// TwinCAT 3 PLC project BohrMachine
// ProgramVersion: 3.1.4023.0
// libraries:
//   Tc2_MC2, * (Beckhoff Automation GmbH)
//   Tc2_Standard, * (Beckhoff Automation GmbH)
//   Tc2_System, * (Beckhoff Automation GmbH)
//   Tc2_Utilities, * (Beckhoff Automation GmbH)
//   Tc3_EventLogger, * (Beckhoff Automation GmbH)
//   Tc3_Module, * (Beckhoff Automation GmbH)
//   VisuSymbols,3.5.10.0,System
// project tree:
//   DUTs/ E_BOHRER_STATES.TcDUT
//   / GlobalTextList.TcGTLO, PlcTask.TcTTO, VisualizationManager.TcVMO (not stored)
//   GVLs/ GVL_Config.TcGVL, GVL_Control.TcGVL
//   POUs/ AxesManager.TcPOU, Bohrkopf.TcPOU, Bohrmaschine.TcPOU, F_Log.TcPOU, I_MachineLogger.TcIO, MachineLogger.TcPOU, MAIN.TcPOU
//   VISUs/ UI.TcVIS
// real-time tasks:
//   TASK PlcTask: cycle T#10ms, priority 20, ADS port 350
//   TASK PlcTask1: cycle T#10ms, priority 21, ADS port 351
//   TASK PlcTask2: cycle T#10ms, priority 22, ADS port 352
//   TASK PlcTask3: cycle T#10ms, priority 23, ADS port 353
//   TASK ControllerTask: cycle T#10ms, priority 1, ADS port 354
//   TASK PlcTask4: cycle T#10ms, priority 24, ADS port 355
//   TASK PlcTask5: cycle T#10ms, priority 25, ADS port 356
// motion (NC):
//   TASK NC-Task 1 SAF: cycle T#2ms, priority 4, ADS port 501
//   TASK NC-Task 1 SVB: cycle T#10ms, priority 8, ADS port 511
//   AXIS xAchse (id 1) // Links-Rechts-Bewegung des Bohrers
//     OtherSettings: AllowMotionCmdToSlave=true
//     encoder EncType=1
//     drive DrvType=5
//       Analog: TorqueSetpointScale=10
//       TimeComp: TaskDelayCycles=1
//     controller CtrType=1
//       CtrPara: PriorControlFactor=1
//         Observer: BandWidth=20
//   AXIS yAchse (id 2) // Hoch-Runter-Bewegung des Bohrers
//     OtherSettings: AllowMotionCmdToSlave=true
//     encoder EncType=1
//     drive DrvType=5
//       Analog: TorqueSetpointScale=10
//       TimeComp: TaskDelayCycles=1
//     controller CtrType=1
//       CtrPara: PriorControlFactor=1
//         Observer: BandWidth=20
//   AXIS zAchse (id 3) // Vor-Zurück-Bewegung des Bohrers
//     OtherSettings: AllowMotionCmdToSlave=true
//     encoder EncType=1
//     drive DrvType=5
//       Analog: TorqueSetpointScale=10
//       TimeComp: TaskDelayCycles=1
//     controller CtrType=1
//       CtrPara: PriorControlFactor=1
//         Observer: BandWidth=20
//   AXIS TransportA (id 4)
//     OtherSettings: AllowMotionCmdToSlave=true
//     encoder EncType=1
//     drive DrvType=5
//       Analog: TorqueSetpointScale=10
//       TimeComp: TaskDelayCycles=1
//     controller CtrType=1
//       CtrPara: PriorControlFactor=1
//         Observer: BandWidth=20
//   AXIS TransportB (id 5)
//     OtherSettings: AllowMotionCmdToSlave=true
//     encoder EncType=1
//     drive DrvType=5
//       Analog: TorqueSetpointScale=10
//       TimeComp: TaskDelayCycles=1
//     controller CtrType=1
//       CtrPara: PriorControlFactor=1
//         Observer: BandWidth=20
// variable links:
//   BohrMachine/BohrMachine Instance <-> Controller/Controller_Obj1 (ModuleController)
//     PlcTask Outputs/MAIN.bohrmaschine.eZustand <-> Bohrmaschine/State
//     PlcTask Outputs/MAIN.bohrmaschine.objID <-> InputIPointers/oidBohrmaschine
//   SuperBohrmachine/SuperBohrmachine Instance <-> NC-Task 1 SAF/Axes/xAchse
//     PlcTask Inputs/MAIN.fbSuperBohrmachine.fbAxesManager.xAchse.NcToPlc <-> Outputs/ToPlc
//     PlcTask Outputs/MAIN.fbSuperBohrmachine.fbAxesManager.xAchse.PlcToNc <-> Inputs/FromPlc
//   SuperBohrmachine/SuperBohrmachine Instance <-> NC-Task 1 SAF/Axes/yAchse
//     PlcTask Inputs/MAIN.fbSuperBohrmachine.fbBohrkopf.axisRef.NcToPlc <-> Outputs/ToPlc
//     PlcTask Outputs/MAIN.fbSuperBohrmachine.fbBohrkopf.axisRef.PlcToNc <-> Inputs/FromPlc
//   SuperBohrmachine/SuperBohrmachine Instance <-> NC-Task 1 SAF/Axes/zAchse
//     PlcTask Inputs/MAIN.fbSuperBohrmachine.fbAxesManager.zAchse.NcToPlc <-> Outputs/ToPlc
//     PlcTask Outputs/MAIN.fbSuperBohrmachine.fbAxesManager.zAchse.PlcToNc <-> Inputs/FromPlc
//   TransportA/TransportA Instance <-> NC-Task 1 SAF/Axes/TransportA
//     PlcTask Inputs/MAIN.fbTransport.axisTransportA.NcToPlc <-> Outputs/ToPlc
//     PlcTask Outputs/MAIN.fbTransport.axisTransportA.PlcToNc <-> Inputs/FromPlc
//   TransportA/TransportA Instance <-> TransportB/TransportB Instance
//     PlcTask Outputs/MAIN.fbTransport.rActVelocity <-> PlcTask Inputs/MAIN.fbTransportSlave.rMasterVelocity
//   TransportA/TransportA Instance <-> Controller/Controller_Obj1 (ModuleController)
//     PlcTask Outputs/MAIN.fbTransport.eZustand <-> TransportA/State
//     PlcTask Outputs/MAIN.fbTransport.objID <-> InputIPointers/oidTransportA
//   TransportB/TransportB Instance <-> NC-Task 1 SAF/Axes/TransportB
//     PlcTask Inputs/MAIN.fbTransportSlave.axisTransportB.NcToPlc <-> Outputs/ToPlc
//     PlcTask Outputs/MAIN.fbTransportSlave.axisTransportB.PlcToNc <-> Inputs/FromPlc
//   TransportB/TransportB Instance <-> Controller/Controller_Obj1 (ModuleController)
//     PlcTask Outputs/MAIN.fbTransportSlave.eZustand <-> TransportB/State
//     PlcTask Outputs/MAIN.fbTransportSlave.fbSensor.bWerkStueckLiegtAn <-> TransportB/WerkstueckLiegtAn
//     PlcTask Outputs/MAIN.fbTransportSlave.objID <-> InputIPointers/oidTransportB

CONFIGURATION BohrMachine
    RESOURCE PLC ON TwinCAT3
        TASK PlcTask(INTERVAL := T#10ms, PRIORITY := 20);
        PROGRAM MAIN WITH PlcTask : MAIN;
    END_RESOURCE
END_CONFIGURATION

// ---- DUTs/E_BOHRER_STATES.TcDUT
{attribute 'qualified_only'}
{attribute 'strict'}
TYPE E_BOHRER_STATES :
(
	eBereit := 0,
	eHerunterfahrend,
	eHochfahrend,
	eUnten,
	eOben,
	eFertig
);
END_TYPE

// ---- GVLs/GVL_Config.TcGVL
{attribute 'qualified_only'}
VAR_GLOBAL
	// Konfiguration
//	stConfig: ST_Config := (rLaenge := 400, rBreite := 300, rDicke := 30);
END_VAR

// ---- GVLs/GVL_Control.TcGVL
{attribute 'qualified_only'}
VAR_GLOBAL
	// UI Command
	bRun: BOOL := FALSE;
	// UI Indicator
	bIsRunning: BOOL := FALSE;
	nProgress: USINT := 0;
	
	// bErrors: BOOL := FALSE;
END_VAR

// ---- POUs/I_MachineLogger.TcIO
INTERFACE I_MachineLogger

METHOD LogBohrung : BOOL
VAR_INPUT
	stPunkt: REFERENCE TO ST_2DPoint;
END_VAR
END_METHOD

METHOD LogPunktAngefahren : BOOL
VAR_INPUT
	stPunkt: REFERENCE TO ST_2DPoint;
END_VAR
END_METHOD

METHOD LogStart : BOOL
VAR_INPUT
END_VAR
END_METHOD

METHOD LogStop : BOOL
VAR_INPUT
END_VAR
END_METHOD

END_INTERFACE

// ---- POUs/MAIN.TcPOU
PROGRAM MAIN
VAR
//	fbLogger: MachineLogger;
	bohrmaschine: Bohrmaschine(sObjectName := 'MAIN.Bohrmaschine');
	
	// just for online testing
	// start-stop trigger
	trigRStart: R_TRIG;
	trigFStop: F_TRIG;
	bStart: BOOL := FALSE;
	stTestConfig: ST_Config := (rLaenge := 400, rBreite := 300, rDicke := 30);
	
END_VAR


// TODO config check

bohrmaschine();

trigRStart(CLK := bStart);
IF trigRStart.Q THEN
	F_Log('starting');
	bohrmaschine.Start(stTestConfig);
//	bohrmaschine.Start();
END_IF

//trigFStop(CLK := bStart);
//IF trigFStop.Q THEN
//	F_Log('stopping');
//	bohrmaschine.Stop();
//END_IF

END_PROGRAM

// ---- POUs/Bohrmaschine.TcPOU
{attribute 'c++_compatible'}
FUNCTION_BLOCK Bohrmaschine EXTENDS TcBaseModuleRegistered IMPLEMENTS I_Bohrmaschine
VAR
	fbLogger: MachineLogger;
	ipLogger: I_MachineLogger;
	bohrer: Bohrkopf;
	axesManager: AxesManager;

	// Zustand der Maschine
	eZustand AT %Q*: E_STATES_BOHRMACHINE := E_STATES_BOHRMACHINE.eWaiting;

	// anzufahrende Punkte
	aPunkte: ARRAY [0..3] OF ST_2DPoint;
	nCurIdx: USINT := 0;
	
	// Hilfsvariablen Visualisierung
	nProgressStep: USINT := 0;

	bRunning: BOOL := FALSE;
	stHomePoint: ST_2DPoint := (x := 0, y := 0);
	
	stConfig: ST_Config;
END_VAR


axesManager();
bohrer();

CASE eZustand OF
	E_STATES_BOHRMACHINE.eWaiting:
		// idle
		
	E_STATES_BOHRMACHINE.ESTARTING:
		Starting();
		
	E_STATES_BOHRMACHINE.eStopped:
		// idle

	E_STATES_BOHRMACHINE.eStopping:
		Stopping();

	E_STATES_BOHRMACHINE.eMoving:
		Moving();

	E_STATES_BOHRMACHINE.eDrilling:
		Drilling();
END_CASE

PROPERTY PUBLIC Config : ST_Config
GET
END_GET
SET
VAR
	rBreite: LREAL;
	rLaenge: LREAL;
	rAbstand: LREAL := 10;
END_VAR
THIS^.stConfig := Config;

rBreite := stConfig.rBreite;
rLaenge := stConfig.rLaenge;

// Punkt 1
aPunkte[0].x := rAbstand;
aPunkte[0].y := rAbstand;

// Punkt 2
aPunkte[1].x := 10;
aPunkte[1].y := rBreite - rAbstand;

// Punkt 3
aPunkte[2].x := rLaenge - rAbstand;
aPunkte[2].y := rBreite - rAbstand;

// Punkt 4
aPunkte[3].x := rLaenge - rAbstand;
aPunkte[3].y := rAbstand;

bohrer.Config REF= stConfig;
END_SET
END_PROPERTY

METHOD PRIVATE Drill : BOOL
eZustand := E_STATES_BOHRMACHINE.eDrilling;
END_METHOD

METHOD PRIVATE Drilling : BOOL
VAR_INPUT
END_VAR
VAR
	bGebohrt: BOOL := FALSE;
END_VAR
// Bohren
bohrer.Bohren(bDone => bGebohrt);
IF(bGebohrt) THEN
	// Progressbar + 1
	GVL_Control.nProgress := GVL_Control.nProgress + 1;
	ipLogger.LogBohrung(axesManager.CurrentPoint);

	MoveNext();
END_IF
END_METHOD

METHOD FB_init : BOOL
VAR_INPUT
	bInitRetains : BOOL; // if TRUE, the retain variables are initialized (warm start / cold start)
	bInCopyCode : BOOL;  // if TRUE, the instance afterwards gets moved into the copy code (online change)
	sObjectName: STRING;
	//ipLogger: I_MachineLogger;
END_VAR
//THIS^.ipLogger := ipLogger;
//SUPER^.FB_init(bInitRetains, bInCopyCode, sObjectName);
THIS^.ipLogger := THIS^.fbLogger;
END_METHOD

METHOD FB_reinit : BOOL
VAR_INPUT
END_VAR
SUPER^.FB_reinit();
END_METHOD

METHOD PRIVATE MoveNext : BOOL
// Nächsten Anfahrtspunkt setzen. Bohrloch oder Home.

// Wenn alle Bohrlöcher abgefahren wurden -> go Home / stop
IF nCurIdx > 3 THEN
	Stop();
ELSE // nächsten Bohrpunkt setzen
	axesManager.Start(aPunkte[nCurIdx]);
	nCurIdx := nCurIdx + 1;	
	eZustand := E_STATES_BOHRMACHINE.eMoving;
END_IF
END_METHOD

METHOD PRIVATE Moving : BOOL
VAR_INPUT
END_VAR

IF axesManager.bPunktAngefahren THEN
	F_Log('Moved To:');
	axesManager.LogAxes();
	axesManager.Stop();
	// Progressbar + 1
	GVL_Control.nProgress := GVL_Control.nProgress + 1;
	
	ipLogger.LogPunktAngefahren(axesManager.CurrentPoint);
	// Achsenbewegungen abgeschlossen, Drill
	Drill();
END_IF
END_METHOD

{attribute 'TcTypeSystem'}
{attribute 'no-analysis'}
{attribute 'c++_compatible'}
{attribute 'minimal_input_size' := '4'}
{attribute 'pack_mode' := '4'}
METHOD PUBLIC Start : HRESULT
VAR_INPUT
	config: REFERENCE TO ST_Config;
END_VAR
CASE eZustand OF
	E_STATES_BOHRMACHINE.EWAITING:
		THIS^.Config := config;
		F_Log('BOHRMASCHINE.Start[eWaiting] called');
		eZustand := E_STATES_BOHRMACHINE.ESTARTING;
		Start := S_PENDING;
		
	E_STATES_BOHRMACHINE.ESTOPPED:
		// fertig
		eZustand := E_STATES_BOHRMACHINE.EWAITING;
		Start := S_OK;
		
	ELSE
		Start := S_PENDING;
END_CASE
END_METHOD

METHOD Starting : BOOL
VAR_INPUT
END_VAR
F_Log('start');
// starten
THIS^.bRunning := TRUE;
GVL_Control.bIsRunning := TRUE;
// Progressbar = 0
GVL_Control.nProgress := 0;
axesManager.Enable(bEnableAxes := TRUE);
ipLogger.LogStart();
MoveNext();
END_METHOD

{attribute 'TcTypeSystem'}
{attribute 'no-analysis'}
{attribute 'c++_compatible'}
{attribute 'minimal_input_size' := '4'}
{attribute 'pack_mode' := '4'}
METHOD PUBLIC Stop : HRESULT
CASE eZustand OF
	E_STATES_BOHRMACHINE.ESTOPPING:
		Stop := S_PENDING;
		
	E_STATES_BOHRMACHINE.EWAITING:
		Stop := S_OK;
		
	E_STATES_BOHRMACHINE.ESTOPPED:
		eZustand := E_STATES_BOHRMACHINE.EWAITING;
		Stop := S_OK;
	
ELSE
	// wenn intern durch Ende gestoppt wurde, benötigt es keinen Stop von aussen
	IF THIS^.bRunning = FALSE THEN
		RETURN;
	END_IF
	
	THIS^.bRunning := FALSE;
	GVL_Control.bRun := FALSE;
	//axesManager.Stop();
	bohrer.Stop();
	eZustand := E_STATES_BOHRMACHINE.eStopping;
	nCurIdx := 0;
	
	Stop := S_PENDING;
END_CASE
END_METHOD

METHOD PRIVATE Stopping : BOOL
VAR
	bBohrerStopped: BOOL := FALSE;
END_VAR
// Warten bis der Bohrkopf oben ist, dann zum Nullpunkt fahren
bohrer.Stopping(bDone => bBohrerStopped);
IF bBohrerStopped THEN
	F_Log('Fahre Home');
	axesManager.Start(stHomePoint);
END_IF

IF axesManager.bPunktAngefahren THEN
	F_Log('Home:');
	axesManager.LogAxes();
	axesManager.Stop();
	eZustand := E_STATES_BOHRMACHINE.eStopped;
	GVL_Control.bIsRunning := FALSE;
	// Progressbar + 1
	GVL_Control.nProgress := 9;
	ipLogger.LogStop();
END_IF
END_METHOD

{attribute 'TcTypeSystem'}
{attribute 'no-analysis'}
{attribute 'c++_compatible'}
{attribute 'minimal_input_size' := '4'}
{attribute 'pack_mode' := '4'}
METHOD TcQueryInterface : HRESULT
VAR_INPUT
	iid	: REFERENCE TO IID;
	pipItf	: POINTER TO PVOID;
END_VAR
VAR
	ipBM: I_Bohrmaschine;
END_VAR
IF GuidsEqual(ADR(iid), ADR(TC_GLOBAL_IID_LIST.IID_I_Bohrmaschine)) THEN
	ipBM := THIS^;
	pipItf^ := ITCUNKNOWN_TO_PVOID(ipBM);
	TcAddRef();
	TcQueryInterface := S_OK;
ELSE
	TcQueryInterface := SUPER^.TcQueryInterface(iid, pipItf);
END_IF
END_METHOD

END_FUNCTION_BLOCK

// ---- POUs/MachineLogger.TcPOU
FUNCTION_BLOCK MachineLogger IMPLEMENTS I_MachineLogger
VAR_INPUT
END_VAR
VAR_OUTPUT
END_VAR
VAR
	fbEventMessage: FB_TcMessage;
	
	// Dauer
	tStart: TIME;
END_VAR

METHOD PUBLIC LogBohrung : BOOL
VAR_INPUT
	stPunkt: REFERENCE TO ST_2DPoint;
END_VAR
VAR
	sPara: STRING;
END_VAR
fbEventMessage.CreateEx(TC_EVENTS.BohrEvents.LochGebohrt, 0);
sPara := CONCAT(CONCAT('x = ', LREAL_TO_STRING(stPunkt.x)), CONCAT(', y = ', LREAL_TO_STRING(stPunkt.y)));
fbEventMessage.ipArguments.AddString(sPara);

fbEventMessage.Send(0);
END_METHOD

METHOD PUBLIC LogPunktAngefahren : BOOL
VAR_INPUT
	stPunkt: REFERENCE TO ST_2DPoint;
END_VAR
VAR
	sPara: STRING;
END_VAR
fbEventMessage.CreateEx(TC_EVENTS.BohrEvents.PunktAngefahren, 0);
sPara := CONCAT(CONCAT('x = ', LREAL_TO_STRING(stPunkt.x)), CONCAT(', y = ', LREAL_TO_STRING(stPunkt.y)));
fbEventMessage.ipArguments.AddString(sPara);
fbEventMessage.Send(0);
END_METHOD

METHOD PUBLIC LogStart : BOOL
fbEventMessage.CreateEx(TC_EVENTS.BohrEvents.MaschineGestartet, 0);
fbEventMessage.Send(0);
tStart := TIME();
END_METHOD

METHOD PUBLIC LogStop : BOOL
VAR
	tDauer: TIME;
	sDauer: STRING(255);
	sParam: STRING;
END_VAR
tDauer := TIME() - tStart;
sDauer := TIME_TO_STRING(tDauer);
fbEventMessage.CreateEx(TC_EVENTS.BohrEvents.MaschineGestoppt, 0);
FindAndDelete(pSrcString := ADR(sDauer), pDeleteString := ADR('T#'), pDstString := ADR(sParam), nDstSize := SIZEOF(sParam));
sParam := CONCAT('Dauer: ', sParam);

fbEventMessage.ipArguments.AddString(sParam);
fbEventMessage.Send(0);
END_METHOD

END_FUNCTION_BLOCK

// ---- POUs/Bohrkopf.TcPOU
FUNCTION_BLOCK FINAL Bohrkopf
VAR
	yAchse: AXIS_REF;
	bYEnabled: BOOL := TRUE;
	rYPos: LREAL := 0;
	rYVelo: LREAL := 10;
	
	// Bohrer ist oder war in der aktiven Phase
	bBohrerAktiv: BOOL := FALSE;
	
	bBohrerMove: BOOL := FALSE;
	bBohrerMoved: BOOL := FALSE;
	
	// MC2 Funktionen
	fbAxisPower: MC_Power;
	fbAxisMove: MC_MoveAbsolute;
	
	// aktueller Zustand des Bohrers
	// TODO Init Methode, auch in Bohrmaschine
	eZustand: E_BOHRER_STATES := E_BOHRER_STATES.eBereit;
	
	stConfig: REFERENCE TO ST_Config;
END_VAR

yAchse.ReadStatus();
fbAxisPower(Axis := yAchse, Enable := bYEnabled, Enable_Positive := bYEnabled, Enable_Negative := bYEnabled);
(*
	Es soll 1cm tief in das Werkstück gebohrt werden.
	Der Abstand zwischen Bohrer und Auflagefläche, auf dem das Werkstück liegt,
	beträgt 5cm.
*)

CASE eZustand OF
	E_BOHRER_STATES.eOben:
		bBohrerMove := FALSE;
		eZustand := E_BOHRER_STATES.eFertig;
		F_Log('Bohrkopf ist oben');
		
	E_BOHRER_STATES.eBereit:
		//F_Log('bereit');
	
	E_BOHRER_STATES.eHochfahrend:
		rYPos := 0;
		bBohrerMove := TRUE;
		//F_Log('hochfahrend');
	
	E_BOHRER_STATES.eHerunterfahrend:
		bBohrerAktiv := TRUE;
		// Abstand + Bohrtiefe (positive Y-Achse zeigt nach unten)
//		rYPos := 50 - GVL_Config.stConfig.rDicke + 10;
		rYPos := 50 - stConfig.rDicke + 10;
		bBohrerMove := TRUE;
		//F_Log('herunterfahrend');
	
	E_BOHRER_STATES.eUnten:
		bBohrerMove := FALSE;
		eZustand := E_BOHRER_STATES.eHochfahrend;
		F_Log('Bohrkopf ist unten');
	
END_CASE

// move according to input
fbAxisMove(
	Axis := yAchse,
	Velocity := rYVelo,
	Execute := bBohrerMove,
	Position := rYPos,
	Done => bBohrerMoved
);

IF bBohrerMoved THEN
	bBohrerMoved := FALSE;
	ADSLOGLREAL(
		msgCtrlMask := ADSLOG_MSGTYPE_HINT,
		msgFmtStr := 'Position Bohrer: %f',
		lrealArg := yAchse.NcToPlc.ActPos
	);

	CASE eZustand OF
		// Bohrer ist hochgefahren -> Zustand 'eOben'
		E_BOHRER_STATES.eHochfahrend:
			eZustand := E_BOHRER_STATES.eOben;
		
		// Bohrer ist heruntergefahren -> Zustand 'eUnten'
		E_BOHRER_STATES.eHerunterfahrend:
			eZustand := E_BOHRER_STATES.eUnten;
	END_CASE
END_IF

METHOD PUBLIC Bohren : BOOL
VAR_OUTPUT
	bDone: BOOL := FALSE;
END_VAR
CASE eZustand OF
	E_BOHRER_STATES.eFertig:
		eZustand := E_BOHRER_STATES.eBereit;
		bDone := TRUE;
		
	E_BOHRER_STATES.eBereit:
		eZustand := E_BOHRER_STATES.eHerunterfahrend;
END_CASE
END_METHOD

PROPERTY PUBLIC Config : REFERENCE TO ST_Config
SET
THIS^.stConfig REF= Config;
END_SET
END_PROPERTY

METHOD PUBLIC Stop : BOOL
// Egal wo der Bohrer ist, er wird als 'unten' markiert und fährt hoch
eZustand := E_BOHRER_STATES.eUnten;
END_METHOD

METHOD PUBLIC Stopping : BOOL
VAR_OUTPUT
	bDone: BOOL;
END_VAR
CASE eZustand OF
	E_BOHRER_STATES.eFertig:
		eZustand := E_BOHRER_STATES.eBereit;
		bDone := TRUE;
		
END_CASE
END_METHOD

END_FUNCTION_BLOCK

// ---- POUs/F_Log.TcPOU
FUNCTION F_Log : BOOL
VAR_INPUT
	msg: STRING;
END_VAR

ADSLOGSTR(
	msgCtrlMask := ADSLOG_MSGTYPE_HINT,
	msgFmtStr := msg,
	strArg := ''
);

END_FUNCTION

// ---- POUs/AxesManager.TcPOU
FUNCTION_BLOCK AxesManager
VAR_INPUT
END_VAR
VAR_OUTPUT
	// am Punkt angekommen
	bPunktAngefahren: BOOL;
END_VAR
VAR
	// Achsen der Maschine (X-Z-Achse)
	xAchse: AXIS_REF;
	zAchse: AXIS_REF;
	
	stPunkt: ST_2DPoint;
	
	// MC2 Funktionen
	fbAxisPowerX: MC_Power;
	fbAxisMoveX: MC_MoveAbsolute;
	
	fbAxisPowerZ: MC_Power;
	fbAxisMoveZ: MC_MoveAbsolute;
	
	// Velocity
	xVelo: LREAL := 100;
	zVelo: LREAL := 100;
	
	bMoveAxes: BOOL := FALSE;
	
	bXMoved: BOOL := FALSE;
	bZMoved: BOOL := FALSE;
END_VAR

xAchse.ReadStatus();
zAchse.ReadStatus();

fbAxisMoveX(Axis := xAchse, Velocity := xVelo, Execute := bMoveAxes, Position := stPunkt.x, Done => bXMoved);
fbAxisMoveZ(Axis := zAchse, Velocity := zVelo, Execute := bMoveAxes, Position := stPunkt.y, Done => bZMoved);

bPunktAngefahren := bXMoved AND bZMoved;

PROPERTY PUBLIC CurrentPoint : REFERENCE TO ST_2DPoint
GET
CurrentPoint REF= stPunkt;
END_GET
END_PROPERTY

METHOD PUBLIC Enable : BOOL
VAR_INPUT
	bEnableAxes: BOOL;
END_VAR
fbAxisPowerX(Axis := xAchse, Enable := bEnableAxes, Enable_Positive := bEnableAxes, Enable_Negative := bEnableAxes);
fbAxisPowerZ(Axis := zAchse, Enable := bEnableAxes, Enable_Positive := bEnableAxes, Enable_Negative := bEnableAxes);
END_METHOD

METHOD PUBLIC LogAxes : BOOL
VAR_INPUT
END_VAR
ADSLOGLREAL(
	msgCtrlMask := ADSLOG_MSGTYPE_HINT,
	msgFmtStr := 'x-Achse: %f',
	lrealArg := xAchse.NcToPlc.ActPos
);

ADSLOGLREAL(
	msgCtrlMask := ADSLOG_MSGTYPE_HINT,
	msgFmtStr := 'z-Achse: %f',
	lrealArg := zAchse.NcToPlc.ActPos
);
END_METHOD

METHOD PUBLIC Start : BOOL
VAR_INPUT
	stPunkt: REFERENCE TO ST_2DPoint;
END_VAR
THIS^.stPunkt := stPunkt;

// quick fix: einmal falsen
fbAxisMoveX(Axis := xAchse, Execute := FALSE);
fbAxisMoveZ(Axis := zAchse, Execute := FALSE);

bMoveAxes := TRUE;
END_METHOD

METHOD PUBLIC Stop : BOOL
VAR_INPUT
END_VAR
bMoveAxes := FALSE;
END_METHOD

END_FUNCTION_BLOCK

// ---- GlobalTextList.TcGTLO
TEXTLIST GlobalTextList
  595 = '%.2f'
  883 = '%2.0f'
  981 = '%2.2f'
  85 = '%f'
  472 = 'Breite'
  473 = 'Breite:'
  136 = 'Dicke:'
  991 = 'Fortschritt'
  426 = 'GVL_'
  487 = 'Konfiguration'
  372 = 'Konfiguration Werkstück'
  701 = 'Länge:'
  507 = 'Start'
  854 = 'Status'
  762 = 'Steuerung'
  956 = 'Stop'
END_TEXTLIST

// ---- VISUs/UI.TcVIS
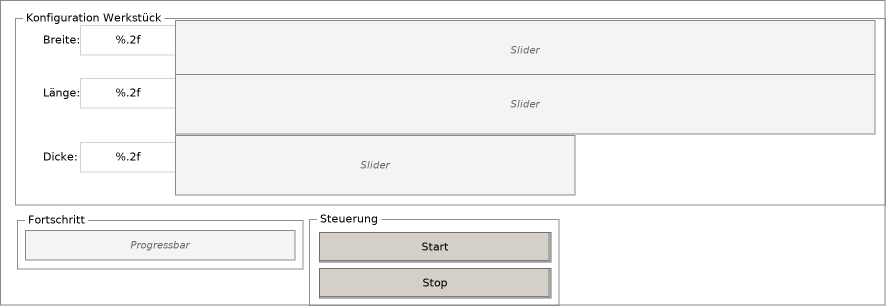
VISUALIZATION UI  // 886x306
    GroupBox (15,10 871x195), "Konfiguration Werkstück", input disabled if: GVL_Control.bIsRunning
        Label (25,15 100x30), "Breite:"
        Label (25,68 100x30), "Länge:"
        Label (25,132 100x30), "Dicke:"
        Textfield (65,15 96x30), "%.2f", text variable: GVL_Config.stConfig.rBreite
        Textfield (65,68 96x30), "%.2f", text variable: GVL_Config.stConfig.rLaenge
        Textfield (65,132 96x30), "%.2f", text variable: GVL_Config.stConfig.rDicke
        Slider (160,10 700x60), variable: GVL_Config.stConfig.rBreite, scale 300..600
        Slider (160,64 700x60), variable: GVL_Config.stConfig.rLaenge, scale 300..600
        Slider (160,125 400x60), variable: GVL_Config.stConfig.rDicke, scale 15..45
    GroupBox (17,212 286x57), "Fortschritt"
        Progressbar (8,18 270x30), variable: GVL_Control.nProgress
    GroupBox (309,211 250x95), "Steuerung"
        Button (10,21 232x30), "Start", input disabled if: GVL_Control.bIsRunning
            OnMouseClick: toggle GVL_Control.bRun
        Button (10,57 232x30), "Stop", input disabled if: (GVL_Control.bIsRunning AND NOT GVL_Control.bRun) OR NOT GVL_Control.bRun
            OnMouseClick: toggle GVL_Control.bRun
END_VISUALIZATION
